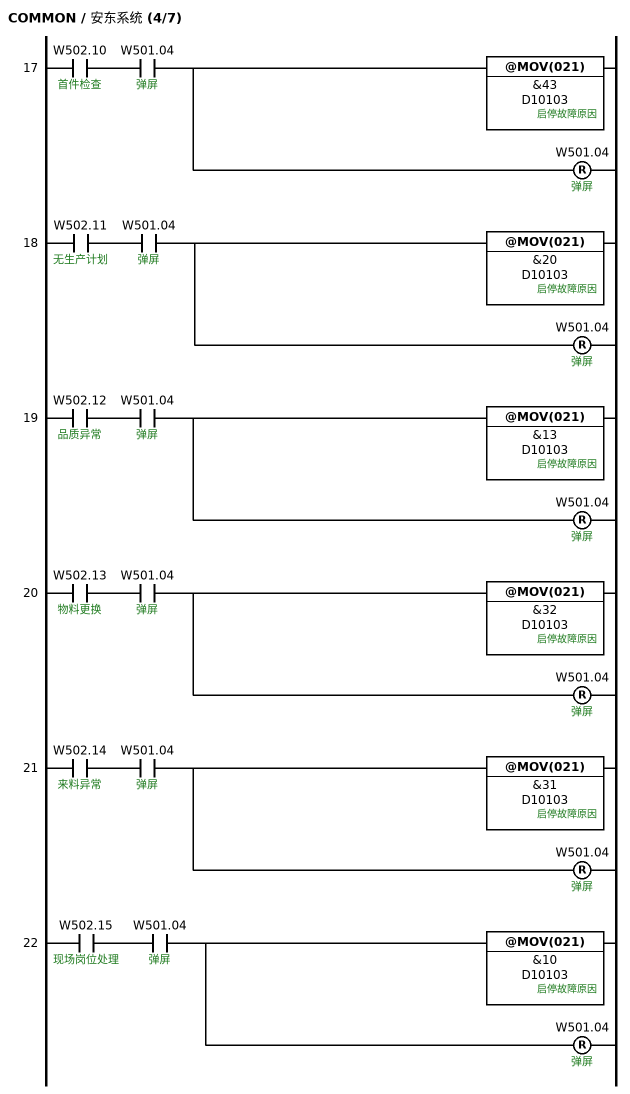
; [picture p480: COMMON / 安东系统, rungs 17-22]
; rung 17
LD W502.10  ; 首件检查
AND W501.04  ; 弹屏
@MOV(021) &43 D10103  ; 启停故障原因
RSET W501.04  ; 弹屏
; rung 18
LD W502.11  ; 无生产计划
AND W501.04  ; 弹屏
@MOV(021) &20 D10103  ; 启停故障原因
RSET W501.04  ; 弹屏
; rung 19
LD W502.12  ; 品质异常
AND W501.04  ; 弹屏
@MOV(021) &13 D10103  ; 启停故障原因
RSET W501.04  ; 弹屏
; rung 20
LD W502.13  ; 物料更换
AND W501.04  ; 弹屏
@MOV(021) &32 D10103  ; 启停故障原因
RSET W501.04  ; 弹屏
; rung 21
LD W502.14  ; 来料异常
AND W501.04  ; 弹屏
@MOV(021) &31 D10103  ; 启停故障原因
RSET W501.04  ; 弹屏
; rung 22
LD W502.15  ; 现场岗位处理
AND W501.04  ; 弹屏
@MOV(021) &10 D10103  ; 启停故障原因
RSET W501.04  ; 弹屏

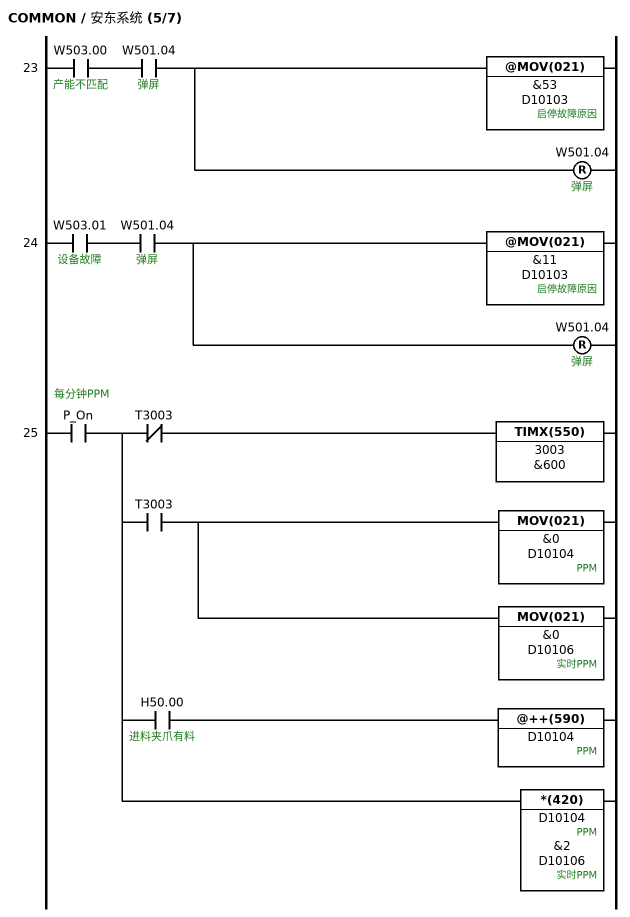
; rung 23
LD W503.00  ; 产能不匹配
AND W501.04  ; 弹屏
@MOV(021) &53 D10103  ; 启停故障原因
RSET W501.04  ; 弹屏
; rung 24
LD W503.01  ; 设备故障
AND W501.04  ; 弹屏
@MOV(021) &11 D10103  ; 启停故障原因
RSET W501.04  ; 弹屏
; rung 25: 每分钟PPM
LD P_On
OUT TR0
ANDNOT T3003
TIMX(550) 3003 &600
LD TR0
AND T3003
MOV(021) &0 D10104  ; PPM
MOV(021) &0 D10106  ; 实时PPM
LD TR0
AND H50.00  ; 进料夹爪有料
@++(590) D10104  ; PPM
LD TR0
*(420) D10104 &2 D10106  ; PPM, 实时PPM

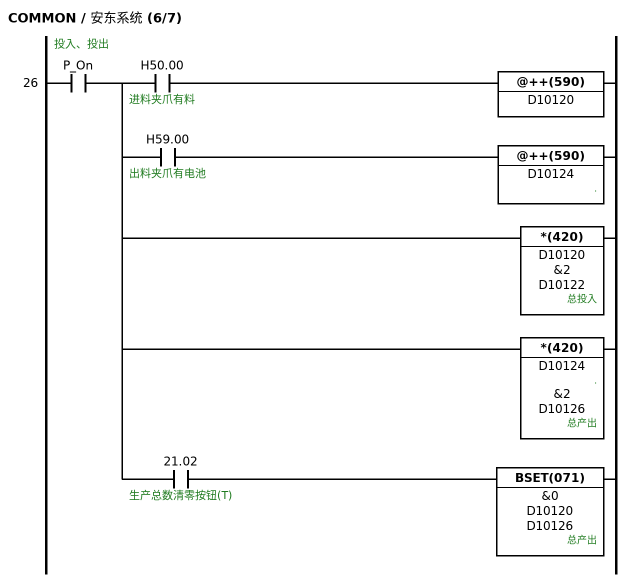
; rung 26: 投入、投出
LD P_On
OUT TR0
AND H50.00  ; 进料夹爪有料
@++(590) D10120
LD TR0
AND H59.00  ; 出料夹爪有电池
@++(590) D10124  ; .
LD TR0
*(420) D10120 &2 D10122  ; 总投入
*(420) D10124 &2 D10126  ; ., 总产出
AND 21.02  ; 生产总数清零按钮(T)
BSET(071) &0 D10120 D10126  ; 总产出

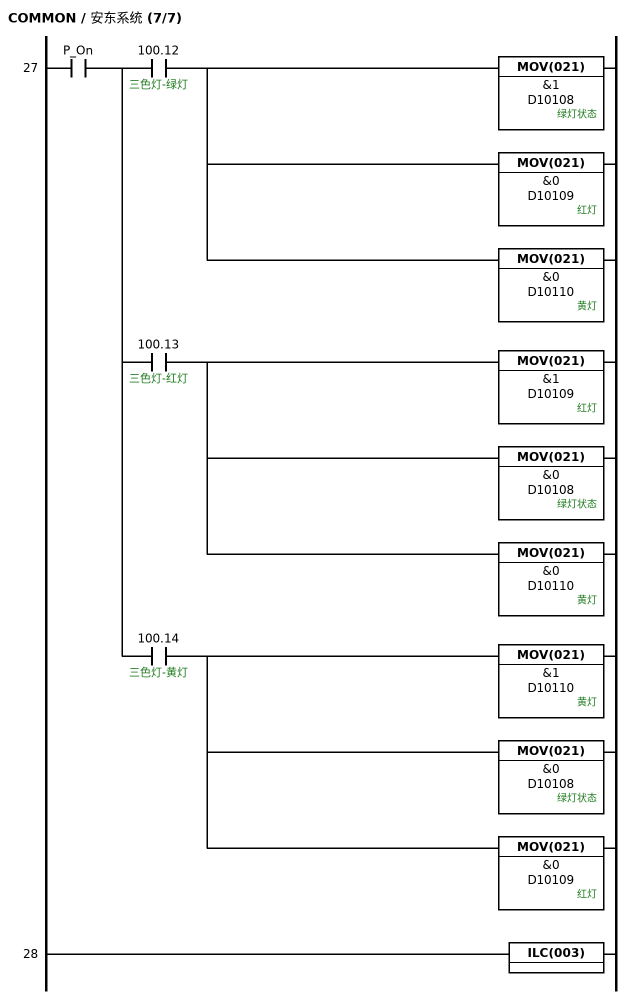
; rung 27
LD P_On
OUT TR0
AND 100.12  ; 三色灯-绿灯
MOV(021) &1 D10108  ; 绿灯状态
MOV(021) &0 D10109  ; 红灯
MOV(021) &0 D10110  ; 黄灯
LD TR0
AND 100.13  ; 三色灯-红灯
MOV(021) &1 D10109  ; 红灯
MOV(021) &0 D10108  ; 绿灯状态
MOV(021) &0 D10110  ; 黄灯
LD TR0
AND 100.14  ; 三色灯-黄灯
MOV(021) &1 D10110  ; 黄灯
MOV(021) &0 D10108  ; 绿灯状态
MOV(021) &0 D10109  ; 红灯
; rung 28
ILC(003)

### Section END
; rung 0
END(001)

## Function block SMC_ISE30A_Convert
VAR_INPUT
  intSensorValue : INT;
END_VAR
VAR_OUTPUT
  fltPressValue : REAL;
END_VAR
VAR
  fltCal_01 : REAL;
  fltCal_02 : REAL;
  fltCal_03 : REAL;
  fltCal_04 : REAL;
  fltInputX : REAL;
  fltXMax : REAL := +4000.0;  (* 模拟量输入最大值 *)
  fltXMin : REAL;  (* 模拟量输入最小值 *)
  ftlYMax : REAL := +1000000.0;  (* 压力表实际最大值1.0MPa *)
  fltYMin : REAL := -100000.0;  (* 压力表实际最小值-0.1MPa *)
  fltCal_05 : REAL;
  fltCal_06 : REAL;
  fltCal_07 : REAL;
END_VAR

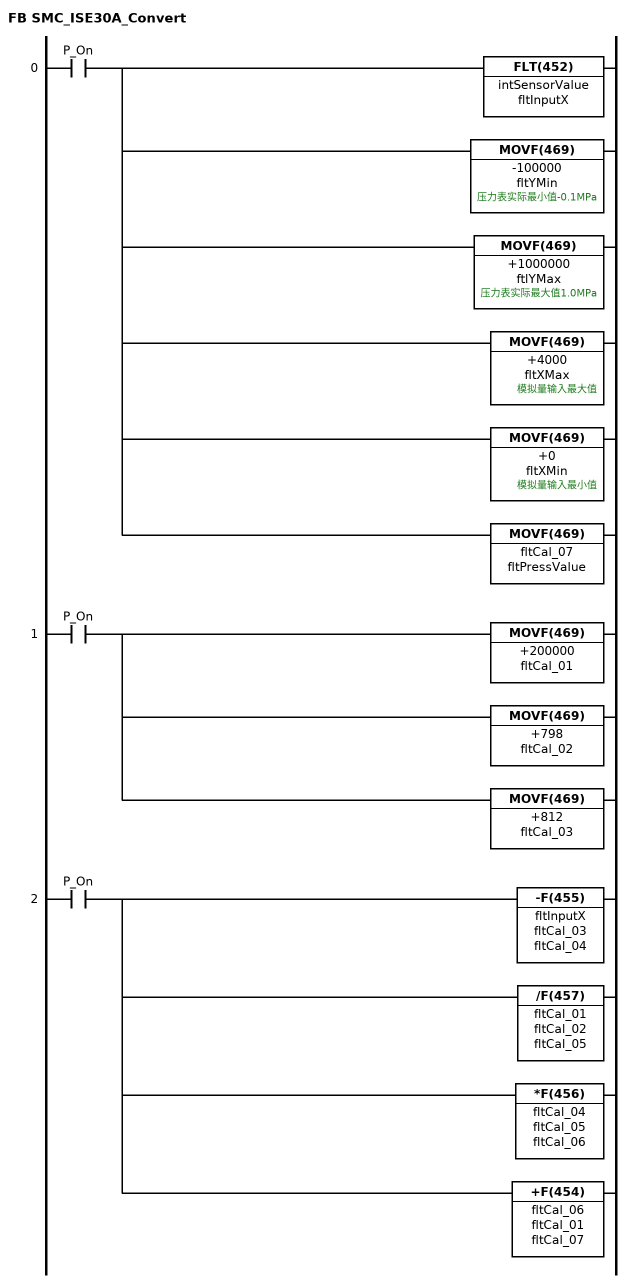
; rung 0
LD P_On
FLT(452) intSensorValue fltInputX
MOVF(469) -100000 fltYMin  ; 压力表实际最小值-0.1MPa
MOVF(469) +1000000 ftlYMax  ; 压力表实际最大值1.0MPa
MOVF(469) +4000 fltXMax  ; 模拟量输入最大值
MOVF(469) +0 fltXMin  ; 模拟量输入最小值
MOVF(469) fltCal_07 fltPressValue
; rung 1
LD P_On
MOVF(469) +200000 fltCal_01
MOVF(469) +798 fltCal_02
MOVF(469) +812 fltCal_03
; rung 2
LD P_On
-F(455) fltInputX fltCal_03 fltCal_04
/F(457) fltCal_01 fltCal_02 fltCal_05
*F(456) fltCal_04 fltCal_05 fltCal_06
+F(454) fltCal_06 fltCal_01 fltCal_07

## Function block VacuumPress_Convert
VAR_INPUT
  intSensorValue : INT;
  fltPressOffset : REAL;  (* 修正值 *)
END_VAR
VAR_OUTPUT
  fltPressValue : REAL;
END_VAR
VAR
  fltCal_01 : REAL;
  fltCal_02 : REAL;
  fltCal_03 : REAL;
  fltCal_04 : REAL;
  fltCal_05 : REAL;
  fltInputX : REAL;
  fltXMax : REAL := +4000.0;  (* 模拟量输入最大值 *)
  fltXMin : REAL;  (* 模拟量输入最小值 *)
  ftlYMax : REAL := +1000000.0;  (* 压力表实际最大值1.0MPa *)
  fltYMin : REAL := -100000.0;  (* 压力表实际最小值-0.1MPa *)
  fltCal_06 : REAL;
  fltCal_07 : REAL;
  fltCal_08 : REAL;
END_VAR

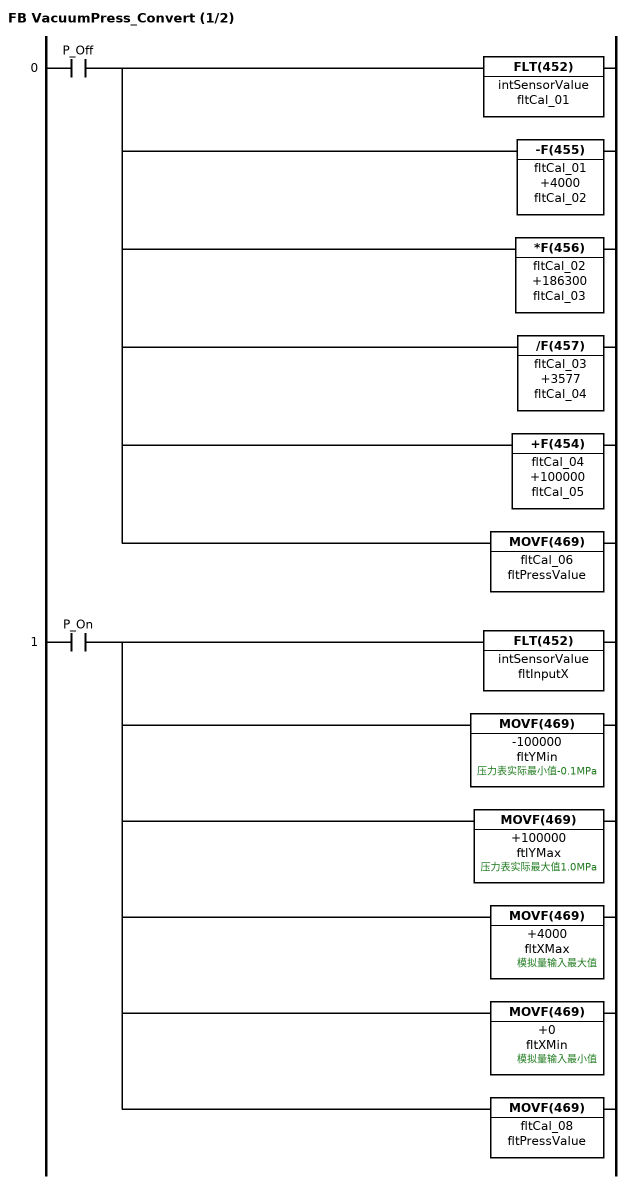
; rung 0
LD P_Off
FLT(452) intSensorValue fltCal_01
-F(455) fltCal_01 +4000 fltCal_02
*F(456) fltCal_02 +186300 fltCal_03
/F(457) fltCal_03 +3577 fltCal_04
+F(454) fltCal_04 +100000 fltCal_05
MOVF(469) fltCal_06 fltPressValue
; rung 1
LD P_On
FLT(452) intSensorValue fltInputX
MOVF(469) -100000 fltYMin  ; 压力表实际最小值-0.1MPa
MOVF(469) +100000 ftlYMax  ; 压力表实际最大值1.0MPa
MOVF(469) +4000 fltXMax  ; 模拟量输入最大值
MOVF(469) +0 fltXMin  ; 模拟量输入最小值
MOVF(469) fltCal_08 fltPressValue

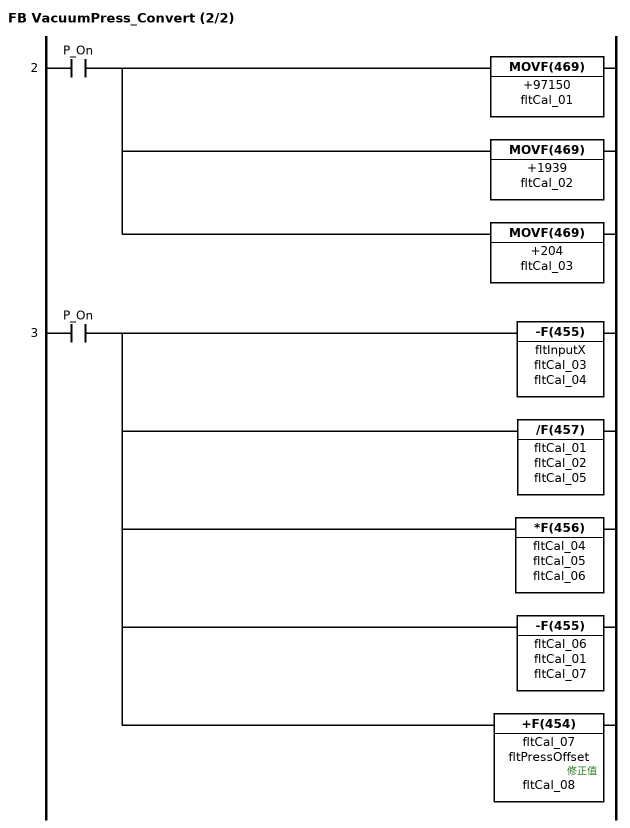
; rung 2
LD P_On
MOVF(469) +97150 fltCal_01
MOVF(469) +1939 fltCal_02
MOVF(469) +204 fltCal_03
; rung 3
LD P_On
-F(455) fltInputX fltCal_03 fltCal_04
/F(457) fltCal_01 fltCal_02 fltCal_05
*F(456) fltCal_04 fltCal_05 fltCal_06
-F(455) fltCal_06 fltCal_01 fltCal_07
+F(454) fltCal_07 fltPressOffset fltCal_08  ; 修正值